// TIA Portal V17 export
// export: Created 2025-03-12T15:36:03.5430515Z, ExportSetting WithDefaults, DisplayName Totally Integrated Automation Portal, DisplayVersion V17 Update 8, DisplayName TIA Portal Openness, DisplayVersion V17 Update 8, DisplayName TIA Portal Version Control Interface, DisplayVersion V17, DisplayName SINAMICS Startdrive Advanced, DisplayVersion V17 SP2, DisplayName SINAMICS Startdrive G110M, G120, G120C, G120D, G120P, G115D, DisplayVersion V17 SP2, DisplayName SINAMICS Startdrive G130, G150, S120, S150, SINAMICS MV, S210, DisplayVersion V17 SP2, DisplayName STEP 7 Professional, DisplayVersion V17 Update 8, DisplayName SINUMERIK ONE STEP 7 Toolbox, DisplayVersion V17 Update 12, DisplayName SINUMERIK 840D sl STEP 7 Toolbox, DisplayVersion V17 Update 12, DisplayName STEP 7 Safety, DisplayVersion V17 Update 6, DisplayName WinCC Advanced, DisplayVersion V17 Update 8
DATA_BLOCK "DB6500_SMC_CYLINDER_HMI"   // DB6500
{ S7_Optimized_Access := 'FALSE'; DB_Accessible_From_OPC_UA := 'FALSE' }
VERSION : 0.1
// stored: AutoNumber false, DBAccessibleFromOPCUA false, DBAccessibleFromWebserver true, IsOnlyStoredInLoadMemory false, IsWriteProtectedInAS false
   VAR
      JXCP_AXIS_HMI_SELECTION : Word := 16#1;   // SELECTED AXIS FOR JXCP1 CONTROLLER
      JXCP_AXIS_MAIN_DB_HMI : Word;   // MAIN SIGNALS SELECTED JXCP1 CONTROLLER
      JXCP_AXIS_AUX_DB_HMI : Word;   // AUX SIGNALS SELECTED JXCP1 CONTROLLER
      LEC_AXIS_HMI_SELECTION : Word := 16#1;   // SELECTED AXIS FOR LECSN CONTROLLER
      LEC_AXIS_CONTROLLER_SIGNALS : Word;   // CONTROLLER SIGNALS
      LEC_AXIS_DATA : Word;   // AXIS DATA
   END_VAR
BEGIN
END_DATA_BLOCK
